Fanuc KAREL source: kd00018.KL

-- PROVISIONAL review KL for V940-1; original PC SHA256 bb32eaac1485fcbb2a6fc38ff3295755847ebe3fbf2e1f37b9fe764f50c3efbc
-- Incomplete behavior may be omitted. Consult companion uncertainty JSON. Do not deploy.
PROGRAM KD00018
%NOLOCKGROUP
VAR
  I : INTEGER
  J : INTEGER
  B : BOOLEAN
  R : REAL
  S : STRING[80]
BEGIN
  -- V9_ZERO_TABLE_METADATA_HINT layout=0001; no indexed target words; source/name/runtime held
  -- UNRESOLVED_PC offsets 5-7; opcodes 9D,4D
  -- UNRESOLVED_PC offsets 12-16; opcodes 7F
END KD00018
